FUNCTION_BLOCK FB_NOT (* Boolean complement *)
  (* Standard: 61499-1-D.1; Classification: Boolean operations *)
  (* Version 0.1, 2001-08-06, JHC, Rockwell Automation, XML version *)
  (* Version 0.0, 1999-02-05, JHC, Rockwell Automation, SRC version *)
  (* Compiler header: package fb.rt.cs725; *)
  (* Compiler classdef: class FB_NOT extends FBFunction1 *)
  (* Compiler Java IBM VisualAge 3.0 *)
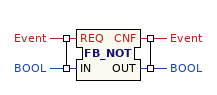
  EVENT_INPUT
    REQ WITH IN;
  END_EVENT
  EVENT_OUTPUT
    CNF WITH OUT;
  END_EVENT
  VAR_INPUT
    IN : BOOL;
  END_VAR
  VAR_OUTPUT
    OUT : BOOL; (* NOT IN *)
  END_VAR
END_FUNCTION_BLOCK
